// TwinCAT 3 PLC project Untitled1
// ProgramVersion: 3.1.4020.4
// libraries:
//   Tc2_MC2, * (Beckhoff Automation GmbH)
//   Tc2_Standard, * (Beckhoff Automation GmbH)
//   Tc2_System, * (Beckhoff Automation GmbH)
//   Tc3_Module, * (Beckhoff Automation GmbH)
// project tree:
//   DUTs/ E_AxisState.TcDUT, ST_Axis.TcDUT
//   GVLs/ IO.TcGVL
//   / PlcTask.TcTTO
//   POUs/ DataProcess.TcPOU, fbAxisControl.TcPOU, MAIN.TcPOU
// real-time tasks:
//   TASK PlcTask: cycle T#10ms, priority 20, ADS port 350
// motion (NC):
//   TASK NC-Task 1 SAF: cycle T#2ms, priority 4, ADS port 501
//   TASK NC-Task 1 SVB: cycle T#10ms, priority 8, ADS port 511
//   AXIS Axis_1 (id 1)
//     General: UnitFlags=#x00000002
//     Dynamic: AccelerationMaximum=0.1, DecelerationMaximum=0.1, Acceleration=0.05, Deceleration=0.05, Jerk=0.1, DelayTime=0.008
//     Velo: Maximum=1.5
//     OtherSettings: AllowMotionCmdToSlave=true
//     encoder EncType=29
//       EncPara: ScaleFactorNumerator=1e-006, ModuloFactor=1, MaxCount=#xffffffff, ReferenceSystem=1
//         Inc: RefSoftSyncMask=#x0000ffff
//     drive DrvType=24
//       Analog: VeloReferenz=2
//       TimeComp: TaskDelayCycles=1
//     controller CtrType=2
//       CtrPara: PriorControlFactor=1
//         PosDiffControl: Range=0.1, Time=0.1
//         PID: PosKp=10, PosExtKp=1
//         Observer: BandWidth=20
// I/O:
//   DEVICE Device 2 (EtherCAT), AmsNetId 198.129.217.73.3.1
//     Term 1 (EK1100) [EK1100 EtherCAT Coupler (2A E-Bus)]
//       Term 2 (EL7031) [EL7031 1Ch. Stepper motor output stage (24V, 1.5A)]
//       Term 3 (EL7031) [EL7031 1Ch. Stepper motor output stage (24V, 1.5A)]
//       Term 4 (EL3202-0010) [EL3202-0010 2Ch. Ana. Input PT100 (RTD), High Precision]
//       Term 5 (EL5002) [EL5002 2Ch. SSI Encoder]
//       Term 6 (EL5042) [EL5042 2Ch. BiSS-C Encoder]
//       Term 16 (EL9011) [EL9011 End Terminal]
//     Term 7 (EK1100) [EK1100 EtherCAT Coupler (2A E-Bus)]
//       Term 8 (EL3102) [EL3102 2Ch. Ana. Input +/-10V, Diff.]
//       Term 9 (EL3602) [EL3602 2Ch. Ana. Input +/-10Volt, Diff. 24bit]
//       Term 10 (EL3602) [EL3602 2Ch. Ana. Input +/-10Volt, Diff. 24bit]
//       Term 11 (EL5101) [EL5101 1Ch. Inc. Encoder 5V]
//       Term 12 (EL3314-0010) [EL3314-0010 4Ch. Ana Input Thermocouple (TC), High Precision]
//       Term 13 (EL9510) [EL9510 Power supply terminal 10V]
//       Term 14 (EL3356-0010) [EL3356-0010 1Ch. Ana. Input Resistor Bridge Terminal, 24bit, High Precision]
//       Term 15 (EL3356-0010) [EL3356-0010 1Ch. Ana. Input Resistor Bridge Terminal, 24bit, High Precision]
//       Term 17 (EL9011) [EL9011 End Terminal]
// variable links:
//   NC-Task 1 SAF/Axes/Axis_1 <-> Device 2 (EtherCAT)/Term 1 (EK1100)/Term 2 (EL7031)
//     Drive/Inputs/In/nState1 @bit 3 <-> STM Status/Status/Error
//     Drive/Inputs/In/nState1 @bit 5 <-> STM Status/Status/Moving negative
//     Drive/Inputs/In/nState1 @bit 4 <-> STM Status/Status/Moving positive
//     Drive/Inputs/In/nState1 @bit 1 <-> STM Status/Status/Ready
//     Drive/Inputs/In/nState1 <-> STM Status/Status/Ready to enable
//     Drive/Inputs/In/nState1 @bit 6 <-> STM Status/Status/Torque reduced
//     Drive/Inputs/In/nState1 @bit 2 <-> STM Status/Status/Warning
//     Drive/Inputs/In/nState2 @bit 3 <-> STM Status/Status/Digital input 1
//     Drive/Inputs/In/nState2 @bit 4 <-> STM Status/Status/Digital input 2
//     Drive/Inputs/In/nState2 @bit 5 <-> STM Status/Status/Sync error
//     Drive/Inputs/In/nState2 @bit 7 <-> STM Status/Status/TxPDO Toggle
//     Drive/Inputs/In/nState4 @bit 1 <-> WcState/InputToggle
//     Drive/Inputs/In/nState4 <-> WcState/WcState
//     Drive/Outputs/Out/nCtrl1 <-> STM Control/Control/Enable
//     Drive/Outputs/Out/nCtrl1 @bit 2 <-> STM Control/Control/Reduce torque
//     Drive/Outputs/Out/nCtrl1 @bit 1 <-> STM Control/Control/Reset
//     Drive/Outputs/Out/nDataOut2[0] <-> STM Velocity/Velocity
//   NC-Task 1 SAF/Axes/Axis_1 <-> Device 2 (EtherCAT)/Term 1 (EK1100)/Term 6 (EL5042)
//     Enc/Inputs/In/nComState @bit 1 <-> WcState/InputToggle
//     Enc/Inputs/In/nComState <-> WcState/WcState
//     Enc/Inputs/In/nDataIn1 <-> FB Inputs Channel 1/Position
//     Enc/Inputs/In/nState1 @bit 12 <-> FB Inputs Channel 1/Status/Diag
//     Enc/Inputs/In/nState1 @bit 1 <-> FB Inputs Channel 1/Status/Error
//     Enc/Inputs/In/nState1 @bit 14 <-> FB Inputs Channel 1/Status/Input cycle counter
//     Enc/Inputs/In/nState1 @bit 2 <-> FB Inputs Channel 1/Status/Ready
//     Enc/Inputs/In/nState1 @bit 13 <-> FB Inputs Channel 1/Status/TxPDO State
//     Enc/Inputs/In/nState1 <-> FB Inputs Channel 1/Status/Warning
//   Untitled1/Untitled1 Instance <-> Device 2 (EtherCAT)/Term 1 (EK1100)/Term 2 (EL7031)
//     PlcTask Inputs/IO.Axis_1.EnableNeg <-> STM Status/Status/Digital input 2
//     PlcTask Inputs/IO.Axis_1.EnablePos <-> STM Status/Status/Digital input 1
//   Untitled1/Untitled1 Instance <-> Device 2 (EtherCAT)/Term 1 (EK1100)/Term 4 (EL3202-0010)
//     PlcTask Inputs/DataProcess.rawRTD <-> RTD Inputs Channel 1/Value
//   Untitled1/Untitled1 Instance <-> Device 2 (EtherCAT)/Term 7 (EK1100)/Term 10 (EL3602)
//     PlcTask Inputs/IO.ai_3_3602 <-> AI Inputs Channel 1/Value
//     PlcTask Inputs/IO.ai_4_3602 <-> AI Inputs Channel 2/Value
//   Untitled1/Untitled1 Instance <-> Device 2 (EtherCAT)/Term 7 (EK1100)/Term 11 (EL5101)
//     PlcTask Inputs/IO.relEnc <-> ENC Status compact/Counter value
//   Untitled1/Untitled1 Instance <-> Device 2 (EtherCAT)/Term 7 (EK1100)/Term 12 (EL3314-0010)
//     PlcTask Inputs/DataProcess.rawTK{1..4} <-> TC Inputs Channel {1..4}/Value  (4 links)
//   Untitled1/Untitled1 Instance <-> Device 2 (EtherCAT)/Term 7 (EK1100)/Term 9 (EL3602)
//     PlcTask Inputs/IO.ai_1_3602 <-> AI Inputs Channel 1/Value
//     PlcTask Inputs/IO.ai_2_3602 <-> AI Inputs Channel 2/Value
//   Untitled1/Untitled1 Instance <-> NC-Task 1 SAF/Axes/Axis_1
//     PlcTask Inputs/IO.Axis_1.Axis.NcToPlc <-> Outputs/ToPlc
//     PlcTask Outputs/IO.Axis_1.Axis.PlcToNc <-> Inputs/FromPlc

CONFIGURATION Untitled1
    RESOURCE PLC ON TwinCAT3
        TASK PlcTask(INTERVAL := T#10ms, PRIORITY := 20);
        PROGRAM MAIN WITH PlcTask : MAIN;
    END_RESOURCE
END_CONFIGURATION

// ---- DUTs/E_AxisState.TcDUT
{attribute 'qualified_only'}
{attribute 'strict'}
TYPE E_AxisState :
(
	INIT := 0,
	READY,
	BUSY,
	ERROR
);
END_TYPE

// ---- DUTs/ST_Axis.TcDUT
TYPE ST_Axis :
STRUCT

(* Input *)
Enable      AT %I*   :   BOOL := TRUE;
EnablePos   AT %I*   :   BOOL := TRUE;
EnableNeg   AT %I*   :   BOOL := TRUE;

DoReset     AT %I*   :   BOOL;
DoHalt      AT %I*   :   BOOL;

SetVelo     AT %I*   :   LREAL := 10;
SetAbsPos   AT %I*   :   LREAL;
DoMoveAbs   AT %I*   :   BOOL;

SetRelDist  AT %I*   :   LREAL;
DoMoveRel   AT %I*   :   BOOL;

(* Output *)
Enabled     AT %Q*   :   BOOL;
Error       AT %Q*   :   BOOL;
LastError   AT %Q*   :   UDINT;
Status      AT %Q*   :   ST_AxisStatus;

(* Internal *)
Axis                 :   AXIS_REF;
State                :   E_AxisState;

END_STRUCT
END_TYPE

// ---- GVLs/IO.TcGVL
{attribute 'qualified_only'}
VAR_GLOBAL
	// *** Axis ***
	Axis_1: ST_Axis;

	// *** Sensor variables ***
	relEnc AT %I* : UINT;
	relPos AT %I* : LREAL;
	
	ai_1_3602 AT %I* : DINT; //Reading from ES3602
	ai_2_3602 AT %I* : DINT; //Reading from ES3602
	ai_3_3602 AT %I* : DINT; //Reading from LV
	ai_4_3602 AT %I* : DINT;
	
	cap3 AT %I*: LREAL; // cap3 reading in um
	cap4 AT %I*: LREAL; // cap4 reading in um
	lv_d AT %I*: LREAL; // laser vibrometer um
	
	motorTemp AT %I* : LREAL; //actuator temp C
	TK1 AT %I* : LREAL;
	TK2 AT %I* : LREAL;
	TK3 AT %I* : LREAL;
	TK4 AT %I* : LREAL;

END_VAR

// ---- POUs/MAIN.TcPOU
PROGRAM MAIN
VAR
	// *** Axis ***
	AxisControl_1: fbAxisControl;

END_VAR

DataProcess();

// *** Axis ***
IF IO.Axis_1.SetVelo = 0 THEN IO.Axis_1.SetVelo := 0.1; END_IF;
AxisControl_1(Axis := IO.Axis_1);

END_PROGRAM

// ---- POUs/fbAxisControl.TcPOU
FUNCTION_BLOCK fbAxisControl
VAR_IN_OUT
	Axis: ST_Axis;
END_VAR
VAR
	mcPower: MC_Power;
	mcReset: MC_Reset;
	mcHalt: MC_Halt;
	mcMoveAbs: MC_MoveAbsolute;
	mcMoveRel: MC_MoveRelative;
END_VAR

(* Update axis status *)
Axis.Axis();

(* Error and Reset transition overrides *)
IF mcReset.Done THEN
    Axis.State := E_AxisState.INIT;
ELSIF Axis.Axis.Status.Error THEN
    Axis.LastError := Axis.Axis.Status.ErrorId;
	Axis.State := E_AxisState.ERROR;
ELSIF mcPower.Error THEN
	Axis.LastError := mcPower.ErrorId;
	Axis.State := E_AxisState.ERROR;
ELSIF mcReset.Error THEN
	Axis.LastError := mcReset.ErrorId;
	Axis.State := E_AxisState.ERROR;
END_IF;


(* Process other state changes *)
CASE Axis.State OF
	
    E_AxisState.INIT :
	Axis.DoReset := FALSE;
	Axis.DoHalt := FALSE;
	Axis.DoMoveAbs := FALSE;
	Axis.DoMoveRel := FALSE;
	Axis.Error := FALSE;
	Axis.LastError := 0;
	Axis.State := E_AxisState.READY;


	E_AxisState.READY :
	IF Axis.Axis.NcToPlc.StateDWord.8 (* HasJob *) THEN
		Axis.State := E_AxisState.BUSY;
    ELSIF mcReset.Busy OR mcHalt.Busy OR mcMoveAbs.Busy OR mcMoveRel.Busy THEN
		Axis.State := E_AxisState.BUSY;
	ELSIF Axis.DoMoveAbs THEN
		mcMoveAbs.Execute := TRUE;
		Axis.State := E_AxisState.BUSY;
	ELSIF Axis.DoMoveRel THEN
		mcMoveRel.Execute := TRUE;
		Axis.State := E_AxisState.BUSY;
	END_IF;

	
	E_AxisState.BUSY :
	(* Move Absolute *)
	Axis.DoMoveAbs := FALSE;
	IF mcMoveAbs.Execute AND NOT mcMoveAbs.Busy THEN
		IF mcMoveAbs.Error THEN
			Axis.LastError := mcMoveAbs.ErrorID;
		ELSIF mcMoveAbs.CommandAborted THEN
			Axis.LastError := 9999;
		ELSIF mcMoveAbs.Done THEN
			Axis.LastError := 0;
		END_IF;
		mcMoveAbs.Execute := FALSE;
	END_IF

	(* Move Relative *)
	Axis.DoMoveRel := FALSE;
	IF mcMoveRel.Execute AND NOT mcMoveRel.Busy THEN
		IF mcMoveRel.Error THEN
			Axis.LastError := mcMoveRel.ErrorID;
		ELSIF mcMoveRel.CommandAborted THEN
			Axis.LastError := 9999;
		ELSIF mcMoveRel.Done THEN
			Axis.LastError := 0;
		END_IF;
		mcMoveRel.Execute := FALSE;
	END_IF

	IF NOT (Axis.Axis.NcToPlc.StateDWord.8 (* HasJob *) OR mcReset.Busy OR mcHalt.Busy OR mcMoveAbs.Busy OR mcMoveRel.Busy) THEN
		Axis.State := E_AxisState.READY;
	END_IF;

	
	E_AxisState.ERROR :
	Axis.Error := TRUE;
	Axis.DoMoveAbs := FALSE;
	Axis.DoMoveRel := FALSE;

END_CASE


(* Execute mothion control function blocks. *)
ActPower();
ActMoveAbs();
ActMoveRel();
ActHalt();
ActReset();

(* Update Axis Status. *)
Axis.Status := Axis.Axis.Status;

ACTION ActHalt:
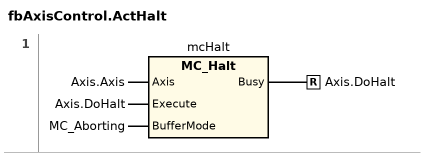
// NETWORK 1
mcHalt(Axis := Axis.Axis, Execute := Axis.DoHalt, BufferMode := MC_Aborting); // MC_Halt
Axis.DoHalt R= mcHalt.Busy;
END_ACTION

ACTION ActMoveAbs:
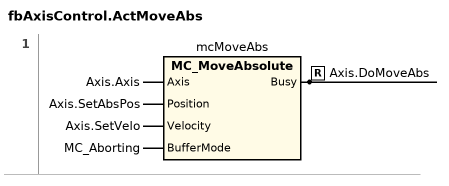
// NETWORK 1
mcMoveAbs(Axis := Axis.Axis, Position := Axis.SetAbsPos, Velocity := Axis.SetVelo, BufferMode := MC_Aborting); // MC_MoveAbsolute
Axis.DoMoveAbs R= mcMoveAbs.Busy;
END_ACTION

ACTION ActMoveRel:
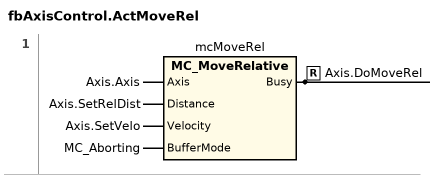
// NETWORK 1
mcMoveRel(
    Axis := Axis.Axis,
    Distance := Axis.SetRelDist,
    Velocity := Axis.SetVelo,
    BufferMode := MC_Aborting); // MC_MoveRelative
Axis.DoMoveRel R= mcMoveRel.Busy;
END_ACTION

ACTION ActPower:
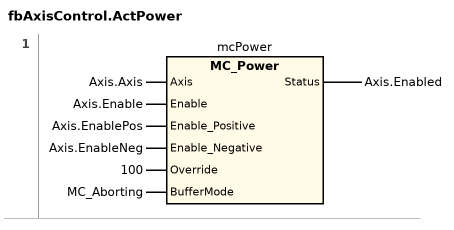
// NETWORK 1
mcPower(
    Axis := Axis.Axis,
    Enable := Axis.Enable,
    Enable_Positive := Axis.EnablePos,
    Enable_Negative := Axis.EnableNeg,
    Override := 100,
    BufferMode := MC_Aborting); // MC_Power
Axis.Enabled := mcPower.Status;
END_ACTION

ACTION ActReset:
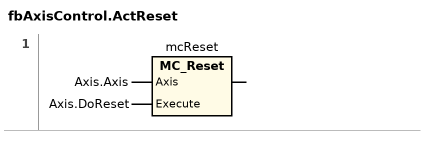
// NETWORK 1
mcReset(Axis := Axis.Axis, Execute := Axis.DoReset); // MC_Reset
END_ACTION

END_FUNCTION_BLOCK

// ---- POUs/DataProcess.TcPOU
PROGRAM DataProcess
VAR
	rawRTD AT %I* : INT;
	
	rawTK1 AT %I* : DINT;
	rawTK2 AT %I* : DINT;
	rawTK3 AT %I* : DINT;
	rawTK4 AT %I* : DINT;
	
END_VAR

IO.relPos := UINT_TO_LREAL(IO.relEnc)*0.1; //um

IO.cap3 := DINT_TO_LREAL(IO.ai_1_3602)*(10.0/2147483648)*(500.0/20.0); //um
IO.cap4 := DINT_TO_LREAL(IO.ai_2_3602)*(10.0/2147483648)*(500.0/20.0); //um
IO.lv_d := DINT_TO_LREAL(IO.ai_3_3602)*(10.0/2147483648)*100 ; //um (100um/V)

IO.motorTemp := INT_TO_LREAL(rawRTD)*0.01; //deg C
IO.TK1 := DINT_TO_LREAL(rawTK1)*0.001; 
IO.TK2 := DINT_TO_LREAL(rawTK2)*0.001;
IO.TK3 := DINT_TO_LREAL(rawTK3)*0.001;
IO.TK4 := DINT_TO_LREAL(rawTK4)*0.001;

END_PROGRAM
